INTERFACE I_HostExtensions EXTENDS __SYSTEM.IQueryInterface

PROPERTY Extensions : I_Extensions
GET
END_GET
END_PROPERTY

END_INTERFACE

(* stored: Version 1.1.0.1, ProductVersion 3.1.4024.12
   Itf I_HostExtensions: Id {b1b6432d-8eed-4ace-82b3-ad4e1dbae0ac}
   Property Extensions: Id {a1047a26-9a42-462d-b26d-b066f3ced646}
   Get Get: Id {d1eff404-b942-4f56-ad60-ead29496521d} *)
